// TIA Portal V21 export
FUNCTION "GestPid_Comando2Valvole" : Void   // FC65, LAD
{ S7_Optimized_Access := 'TRUE' }
// stored: SetENOAutomatically false
   VAR_INPUT
      K_Valvola1 : Int;
      K_Valvola2 : Int;
      K_TipoAccoppiamentoUscitePid : Int;
      K_Pid : Int;
   END_VAR
BEGIN

REGION Network 1 (SCL)
   "Pid".P[#K_Pid].In.K_Valvola1 := #K_Valvola1;
   "Pid".P[#K_Pid].In.K_Valvola2 := #K_Valvola2;
   "Pid".P[#K_Pid].Prm.K_TipoAccoppiamentoUscitePid := #K_TipoAccoppiamentoUscitePid;
END_REGION
END_FUNCTION
